FUNCTION_BLOCK FB_CommandChangeClear EXTENDS FB_CommandChange IMPLEMENTS ITF_CommandChange
VAR

END_VAR

(*			
	RafalOS
	Rafał Osajda		03.11.2025		TC 4024.66
	Test czy można zmienić stan lub tryb i zwraca czy można i uruchamia zmianę
*)
METHOD PUBLIC Execute : BOOL
VAR_INPUT
	iNumberOfCommand	: INT;
END_VAR
IF (THIS^.itfSaMController.GetState () = E_BaseMachineState.Aborted) THEN		// sprawdzenie czy jesteśmy w dobrym stanie dla tego rozkazu
	IF (THIS^.itfSaMController.IsStateInModeEnabled (eState := E_BaseMachineState.Clearing)) THEN	//test czy stan do którego chcemy przejśc jest właczony dla tego trybu
		THIS^.itfSaMController.ChangeStateTo (eNewState := E_BaseMachineState.Clearing);
	ELSE
		THIS^.EventSetActive (iNumber := 5);	//stan docelowy jest wylaczony w tym trybie
	END_IF
ELSE
	THIS^.EventSetActive (iNumber := 4);	//ten rozkaz nie obsluguje tego stanu
END_IF
END_METHOD

METHOD FB_init : BOOL
VAR_INPUT
	bInitRetains : BOOL; // if TRUE, the retain variables are initialized (warm start / cold start)
	bInCopyCode : BOOL;  // if TRUE, the instance afterwards gets moved into the copy code (online change)
END_VAR
THIS^.SetText (eLocation := E_BaseLocation.pl, wsDescription := "Command change state - Clear");
THIS^.SetText (eLocation := E_BaseLocation.en, wsDescription := "Command change state - Clear");
THIS^.SetText (eLocation := E_BaseLocation.de, wsDescription := "Command change state - Clear");
THIS^.SetName (stName := THIS^.GetTexts ());
END_METHOD

END_FUNCTION_BLOCK

(* stored: Version 1.1.0.1
   POU FB_CommandChangeClear: Id {a2f054b4-2db6-03dd-29ad-ebaea950569c}, SpecialFunc None
   Method Execute: Id {e270a742-df07-0314-14d2-7048e77ad1f5}
   Method FB_init: Id {a7563e04-2507-0766-224d-d9198b48a6cb} *)
